PROGRAM progServoCntrl
VAR
	Servo_04_0100 : fbServo;
	
END_VAR

END_PROGRAM

(* stored: Version 1.1.0.1, ProductVersion 3.1.4024.6
   POU progServoCntrl: Id {20ecc3a3-62da-48f6-83ad-2767f7bd919b}, SpecialFunc None *)
